FUNCTION_BLOCK fb_sv_controller
VAR_IN_OUT
	var_ref_sv : ref_sv_io;
END_VAR
VAR_INPUT
	in_flg_run : BOOL;
	in_var_moveMode : eP_svMoveMode;
	in_var_sensorDelay : TIME;
END_VAR
VAR_OUTPUT
	out_flg_run : BOOL;
	out_flg_busy: BOOL;
	out_flg_Done: BOOL;
	out_flg_error : BOOL;
END_VAR
VAR
	var_buf_moveMode: eP_svMoveMode;
	fbi_sensorDelayTimerA: TON;
	fbi_sensorDelayTimerB: TON;
	flg_svADone: BOOL;
	flg_svBDone: BOOL;
	fbi_timeOut: TON;
	flg_svSDone: BOOL;
END_VAR
VAR // added by the converter: edge detectors and wires of the graphical bodies
    _rt1, _rt2, _rt3, _rt4 : R_TRIG;
    _w1, _w2, _w3 : BOOL;
END_VAR

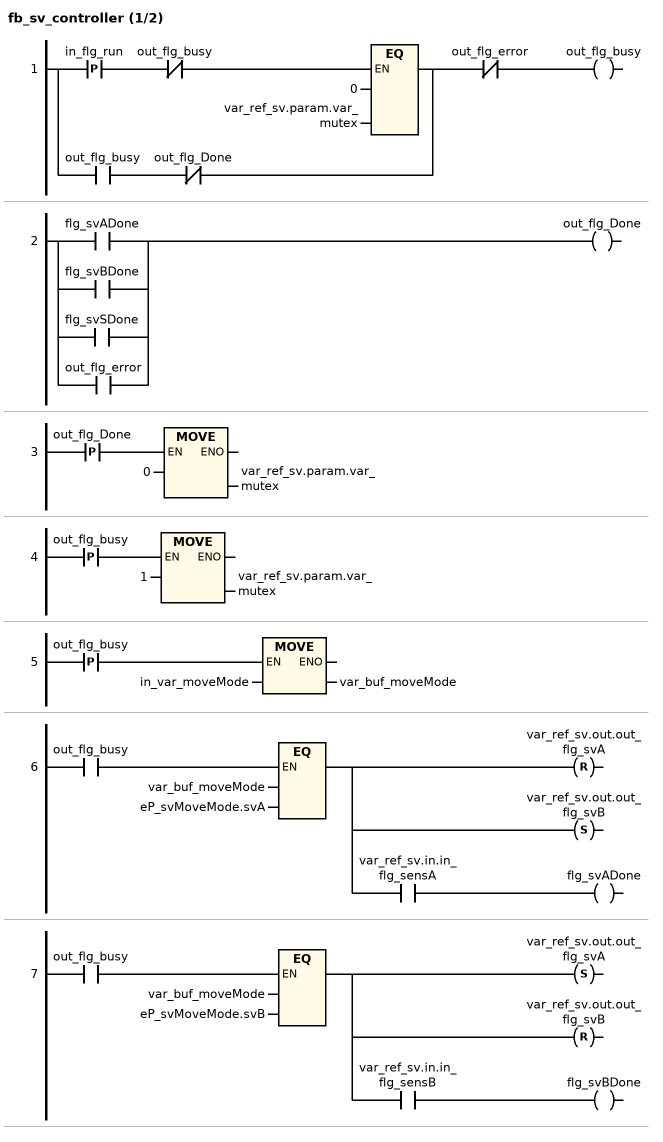
// NETWORK 1
_rt1(CLK := in_flg_run);
out_flg_busy := (_rt1.Q AND NOT out_flg_busy AND 0 = var_ref_sv.param.var_mutex OR out_flg_busy AND NOT out_flg_Done) AND NOT out_flg_error;

// NETWORK 2
out_flg_Done := flg_svADone OR flg_svBDone OR flg_svSDone OR out_flg_error;

// NETWORK 3
_rt2(CLK := out_flg_Done);
IF _rt2.Q THEN var_ref_sv.param.var_mutex := 0; END_IF

// NETWORK 4
_rt3(CLK := out_flg_busy);
IF _rt3.Q THEN var_ref_sv.param.var_mutex := 1; END_IF

// NETWORK 5
_rt4(CLK := out_flg_busy);
IF _rt4.Q THEN var_buf_moveMode := in_var_moveMode; END_IF

// NETWORK 6
_w1 := out_flg_busy AND var_buf_moveMode = eP_svMoveMode.svA;
var_ref_sv.out.out_flg_svA R= _w1;
var_ref_sv.out.out_flg_svB S= _w1;
flg_svADone := _w1 AND var_ref_sv.in.in_flg_sensA;

// NETWORK 7
_w2 := out_flg_busy AND var_buf_moveMode = eP_svMoveMode.svB;
var_ref_sv.out.out_flg_svA S= _w2;
var_ref_sv.out.out_flg_svB R= _w2;
flg_svBDone := _w2 AND var_ref_sv.in.in_flg_sensB;

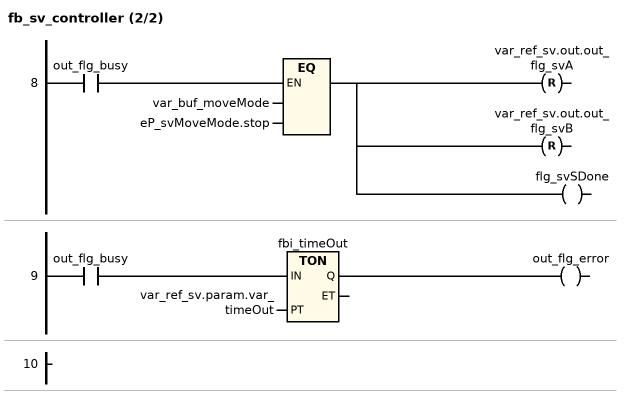
// NETWORK 8
_w3 := out_flg_busy AND var_buf_moveMode = eP_svMoveMode.stop;
var_ref_sv.out.out_flg_svA R= _w3;
var_ref_sv.out.out_flg_svB R= _w3;
flg_svSDone := _w3;

// NETWORK 9
fbi_timeOut(IN := out_flg_busy, PT := var_ref_sv.param.var_timeOut); // TON
out_flg_error := fbi_timeOut.Q;

// NETWORK 10

END_FUNCTION_BLOCK

(* stored: Version 1.1.0.1, ProductVersion 3.1.4024.12
   POU fb_sv_controller: Id {0973bc12-ef64-43d3-890e-b82fee1183c4}, SpecialFunc None *)
